TYPE E_TunerState :
(
    eIdle := 0,
    eReadInductance,
    eReadMaxCurrent,
    eWriteMaxCurrent,
    eCalcStartKp,
    eWriteKp,
    eWriteKi,
    eWaitTnCalc,
    eReadTn,
    eEvaluateTn,
    eMoveFwd,
    eWaitMoveFwd,
    eMoveBwd,
    eWaitMoveBwd,
    eEvaluateResonance,
    eWaitNextStep,
    eApplyBestParams,
    // Manual Param Application
    eApplyManualCurrent,
    eApplyManualKp,
    eApplyManualKi,
    eError
);
END_TYPE

(* stored: Version 1.1.0.1
   DUT E_TunerState: Id {57895a33-eccf-4c2a-8344-d1fdb23c2158} *)
